// Mitsubishi GX Works2 project: master   PLC: Q00

// global labels: Global1
VAR_GLOBAL
  tank_glob AT D0 : INT;
  flow_glob AT D10 : INT;  (* generelt pådrag *)
  pådrag_glob AT D12 : INT;
  organ_glob AT M23 : BOOL;  (* frekvensomformer eller ventil *)
  FO_flow_glob AT D11 : INT;  (* pådrag fra frekvensomformer *)
  slider_glob AT D20 : INT;  (* settverdi *)
  kp_hmi AT D14 : INT;
  ki_hmi AT D15 : INT;
  kd_hmi AT D16 : INT;
  manuell_hmi AT M24 : BOOL;
  tf_hmi AT D17 : INT;
  ventil_1_glob AT M20 : BOOL;
  ventil_2_glob AT M21 : BOOL;
  ventil_3_glob AT M22 : BOOL;
  TIL_FRA_SLAVE_1 : TIL_FRA_SLAVE;
  bResetAlarm_glob AT M25 : BOOL;
  bAlarmCritLow_glob AT M26 : BOOL;
  bAlarmLow_glob AT M27 : BOOL;
  bAlarmHigh_glob AT M28 : BOOL;
  bAlarmCritHigh_glob AT M29 : BOOL;
  bEmergency_glob AT M30 : BOOL;
  iP_glob AT D18 : INT;
  iI_glob AT D19 : INT;
  iD_glob AT D21 : INT;
  auto_iP_glob AT D22 : INT;
  auto_iI_glob AT D23 : INT;
  auto_iD_glob AT D24 : INT;
  auto_Tf_glob AT D25 : INT;
  Start : BOOL;
END_VAR

PROGRAM POU_01
(* structured ladder/FBD written out as ST: instructions are called as NAME(EN, inputs, outputs); _pN, _eN, _tN stand for wires *)
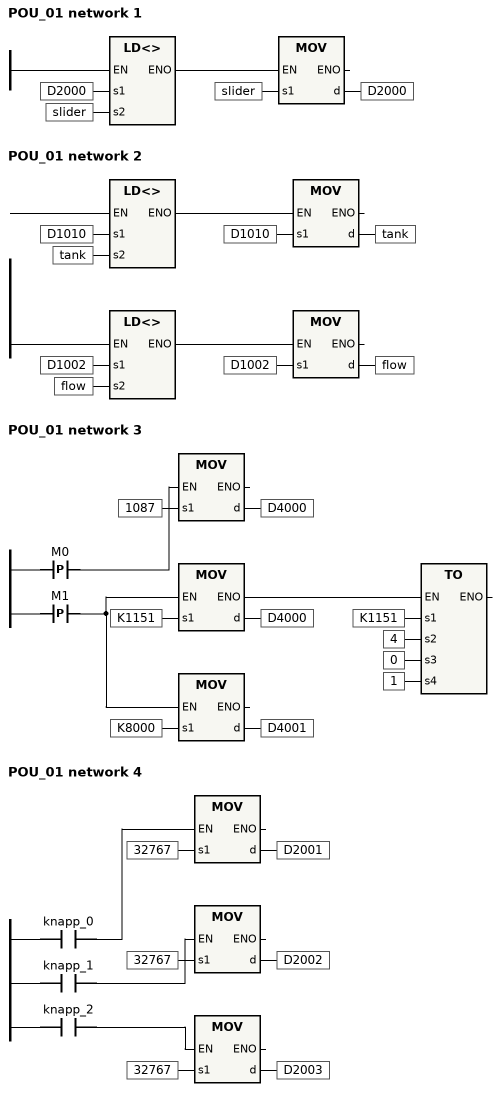
(* network 1 *)
_e1 := LD<>(TRUE, D2000, slider);
MOV(_e1, slider, D2000);
(* network 2 *)
_e1 := LD<>(TRUE, D1010, tank);
MOV(_e1, D1010, tank);
_e2 := LD<>(TRUE, D1002, flow);
MOV(_e2, D1002, flow);
(* network 3 *)
MOV(LDP(TRUE, M0), 1087, D4000);
_p1 := LDP(TRUE, M1);
_e2 := MOV(_p1, K1151, D4000);
TO(_e2, K1151, 4, 0, 1);
MOV(_p1, K8000, D4001);
(* network 4 *)
MOV(knapp_0, 32767, D2001);
MOV(knapp_1, 32767, D2002);
MOV(knapp_2, 32767, D2003);
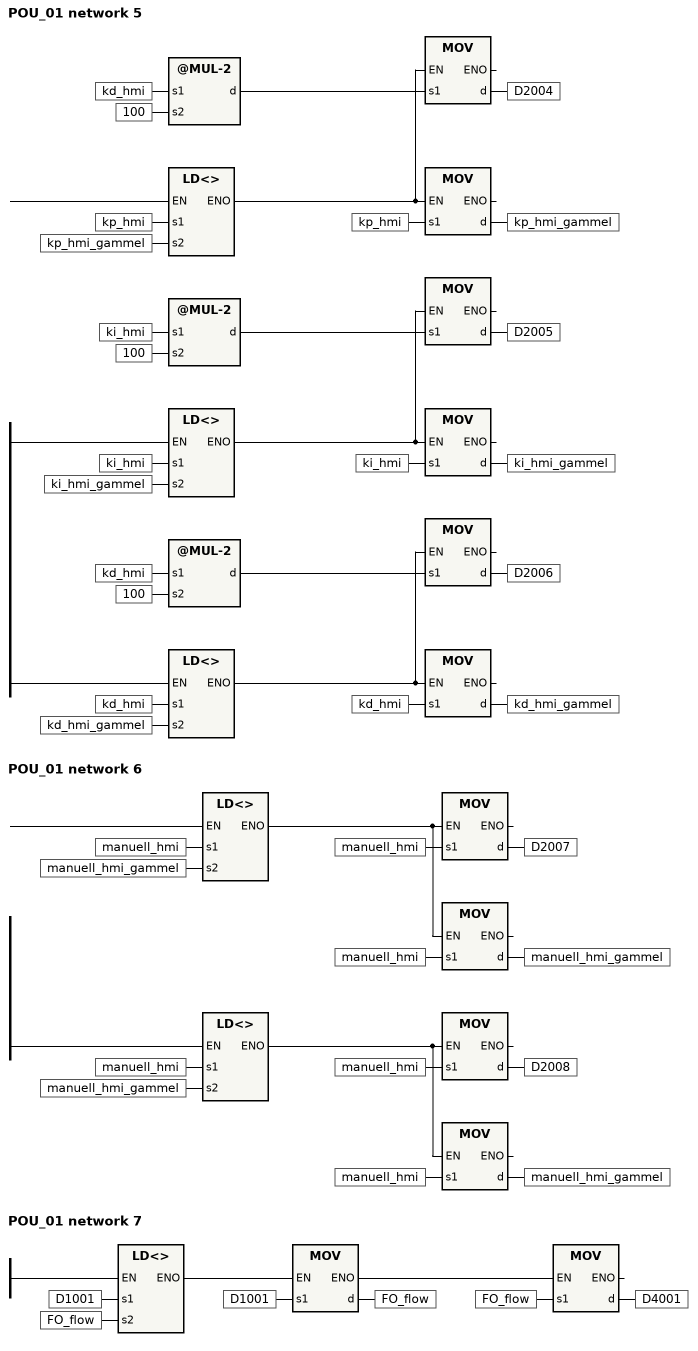
(* network 5 *)
_e1 := LD<>(TRUE, kp_hmi, kp_hmi_gammel);
MOV(_e1, @MUL-2(kd_hmi, 100), D2004);
MOV(_e1, kp_hmi, kp_hmi_gammel);
_e2 := LD<>(TRUE, ki_hmi, ki_hmi_gammel);
MOV(_e2, @MUL-2(ki_hmi, 100), D2005);
MOV(_e2, ki_hmi, ki_hmi_gammel);
_e3 := LD<>(TRUE, kd_hmi, kd_hmi_gammel);
MOV(_e3, @MUL-2(kd_hmi, 100), D2006);
MOV(_e3, kd_hmi, kd_hmi_gammel);
(* network 6 *)
_e1 := LD<>(TRUE, manuell_hmi, manuell_hmi_gammel);
MOV(_e1, manuell_hmi, D2007);
MOV(_e1, manuell_hmi, manuell_hmi_gammel);
_e2 := LD<>(TRUE, manuell_hmi, manuell_hmi_gammel);
MOV(_e2, manuell_hmi, D2008);
MOV(_e2, manuell_hmi, manuell_hmi_gammel);
(* network 7 *)
_e1 := LD<>(TRUE, D1001, FO_flow);
_e2 := MOV(_e1, D1001, FO_flow);
MOV(_e2, FO_flow, D4001);
END_PROGRAM

FUNCTION_BLOCK toggle_hmi
VAR_INPUT
  Input : BOOL;
END_VAR
VAR_OUTPUT
  FlipFlop : BOOL;
END_VAR
VAR
  OldInput : BOOL;
  oneshot : BOOL;
END_VAR
oneshot:= Input AND NOT OldInput;

IF oneshot THEN
	FlipFlop := NOT FlipFlop;
END_IF;

OldInput:=Input;
END_FUNCTION_BLOCK

FUNCTION_BLOCK TIL_FRA_SLAVE
VAR_INPUT
  slider : INT;
END_VAR
VAR_OUTPUT
  tank : INT;
  flow : INT;
END_VAR
VAR_INPUT
  ventil_1 : BOOL;
  ventil_2 : BOOL;
  ventil_3 : BOOL;
  kp : INT;
  ki : INT;
  kd : INT;
  tf : INT;
END_VAR
VAR_OUTPUT
  pådrag : INT;
END_VAR
VAR_INPUT
  organ : BOOL;
  manuell : BOOL;
END_VAR
VAR_OUTPUT
  FO_flow : INT;
END_VAR
VAR
  kp_old : INT;
  ki_old : INT;
  kd_old : INT;
  pådrag_old : INT;
  tf_old : INT;
END_VAR
VAR_OUTPUT
  iP : INT;
  iI : INT;
  iD : INT;
  bAlarmCritLow : BOOL;
  bAlarmLow : BOOL;
  bAlarmHigh : BOOL;
  bAlarmCritHigh : BOOL;
  bEmergency : BOOL;
END_VAR
VAR_INPUT
  bResetAlarm : BOOL;
END_VAR
VAR_OUTPUT
  auto_iP : INT;
  auto_iI : INT;
  auto_iD : INT;
  auto_Tf : INT;
END_VAR
VAR
  TankNy : INT;
  iAlarmWord : INT;
END_VAR
(* ===================== TIL SLAVE===================== *)

(* Referanse *)
MOV(TRUE, slider, D2000);

(* Ventil 1 *)
IF ventil_1 THEN
	MOV(TRUE, 32767, D2001);
ELSE
	MOV(TRUE, 0, D2001);
END_IF;

(* Ventil 2 *)
IF ventil_2 THEN
	MOV(TRUE, 32767, D2002);
ELSE
	MOV(TRUE, 0, D2002);
END_IF;

(* Ventil 3 *)
IF ventil_3 THEN
	MOV(TRUE, 32767, D2003);
ELSE
	MOV(TRUE, 0, D2003);
END_IF;

(* Kp *)
IF kp <> kp_old THEN
	MOV(TRUE, kp, D2004);
	MOV(TRUE, kp, kp_old);
END_IF;

(* Ki *)
IF ki <> ki_old THEN
	MOV(TRUE, ki, D2005);
	MOV(TRUE, ki, ki_old);
END_IF;

(* Kd *)
IF kd <> kd_old THEN
	MOV(TRUE, kd, D2006);
	MOV(TRUE, kd, kd_old);
END_IF;

(* Manuell input*)
IF pådrag <> pådrag_old THEN
	MOV(TRUE, pådrag, D2007);
	MOV(TRUE, pådrag, pådrag_old);
END_IF;

(* Tf *)
IF tf <> tf_old THEN
	MOV(TRUE, tf, D2008);
	MOV(TRUE, tf, tf_old);
END_IF;	

(* Frekvensomformer eller ventil *)
IF organ THEN
	MOV(TRUE, 32767, D2009);
ELSE
	MOV(TRUE, 0, D2009);
END_IF;

(* Manuell eller auto modus *)
IF manuell THEN
	MOV(TRUE, 32767, D2010);
ELSE
	MOV(TRUE, 0, D2010);
END_IF;

(* Kvittering av alarm *)
IF bResetAlarm THEN
    MOV(TRUE, 32767, D2020);
ELSE
    MOV(TRUE, 0, D2020);
END_IF;

(* Autotuning *)
MOV(TRUE, D26, D2012);

(* Nom Pådrag *)
MOV(TRUE, D27, D2013);

(* Foroverkoblingskoeffisient *)
MOV(TRUE, D28, D2014);

(* ===================== FRA SLAVE===================== *)

(* Tank-nivå *)
TankNy := D1010;

IF TankNy > 0 THEN
    IF ABS(TankNy - tank) < 500 OR tank = 0 THEN
        tank := TankNy;
    END_IF;
END_IF;

(* Pådrag *)
MOV(TRUE, D1002, flow);
	
(* Frekvensomformer pådrag *)
IF D1003 <> FO_flow THEN
	MOV(TRUE, D1003, FO_flow);
	MOV(TRUE, FO_flow, D4001);
END_IF;

(* Pådrag Kp *)
IF D1004 <> iP THEN
	MOV(TRUE, D1004, iP);
END_IF;

(* Pådrag Ki *)
IF D1005 <> iI THEN
	MOV(TRUE, D1005, iI);
END_IF;

(* Pådrag Kd *)
IF D1006 <> iD THEN
	MOV(TRUE, D1006, iD);
END_IF;

(* Alarm  *)
bAlarmCritLow  := D1007.0;
bAlarmLow      := D1007.1;
bAlarmCritHigh := D1007.2;
bAlarmHigh     := D1007.3;
bEmergency     := D1007.4;
	
(* Fra autotuning *)
IF D1011 <> auto_iP THEN
	MOV(TRUE, D1011, auto_iP);
END_IF;

IF D1012 <> auto_iI THEN
	MOV(TRUE, D1012, auto_iI);
END_IF;

IF D1013 <> auto_iD THEN
	MOV(TRUE, D1013, auto_iD);
END_IF;

IF D1014 <> auto_Tf THEN
	MOV(TRUE, D1014, auto_Tf);
END_IF;
END_FUNCTION_BLOCK

PROGRAM Master_Main
(* structured ladder/FBD written out as ST: instructions are called as NAME(EN, inputs, outputs); _pN, _eN, _tN stand for wires *)
(* Initialisering *)
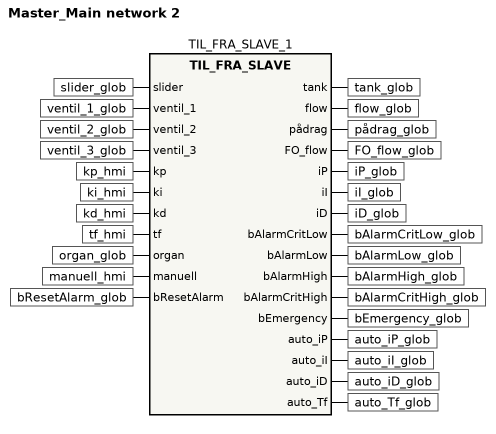
(* network 2 *)
TIL_FRA_SLAVE_1(slider := slider_glob, ventil_1 := ventil_1_glob, ventil_2 := ventil_2_glob, ventil_3 := ventil_3_glob, kp := kp_hmi, ki := ki_hmi, kd := kd_hmi, tf := tf_hmi, organ := organ_glob, manuell := manuell_hmi, bResetAlarm := bResetAlarm_glob, tank => tank_glob, flow => flow_glob, pådrag => pådrag_glob, FO_flow => FO_flow_glob, iP => iP_glob, iI => iI_glob, iD => iD_glob, bAlarmCritLow => bAlarmCritLow_glob, bAlarmLow => bAlarmLow_glob, bAlarmHigh => bAlarmHigh_glob, bAlarmCritHigh => bAlarmCritHigh_glob, bEmergency => bEmergency_glob, auto_iP => auto_iP_glob, auto_iI => auto_iI_glob, auto_iD => auto_iD_glob, auto_Tf => auto_Tf_glob);
END_PROGRAM

FUNCTION_BLOCK INITIERING
VAR_INPUT
  START : BOOL;
END_VAR
MOV(START, 1087, D4000);
END_FUNCTION_BLOCK
